(* IEC 61131-3 sources: xPLCCore/codesys_code/Application/COMM_FBs/FB_DataBuffer, 13 files *)

(* ---- FB_DataBuffer.st ---- *)
(*
    FUNCTION_BLOCK FB_DataBuffer

    A re-usable data buffer that operates on an externally provided BYTE array.
    It provides methods for managing a continuous stream of bytes in that external memory.
*)
FUNCTION_BLOCK FB_DataBuffer

VAR
    (* Internal pointers and size information *)
    pBuffer : POINTER TO BYTE; (* Pointer to the start of the external buffer *)
    udiCapacity :DINT;       (* The logical capacity of the external buffer *)
    udiCurrentSize : DINT := 0; (* The current number of valid bytes in the buffer *)
END_VAR
(* =========== IMPLEMENTATION =========== *)

(* ---- get_buffer.st ---- *)
METHOD get_buffer : POINTER TO BYTE
(* =========== IMPLEMENTATION =========== *)
IF pBuffer <> 0 THEN
    get_buffer := pBuffer;
ELSE
    // If the buffer has not been reset, return a NULL pointer.
    get_buffer := 0;
END_IF

(* ---- get_head.st ---- *)
METHOD get_head : POINTER TO BYTE
(* =========== IMPLEMENTATION =========== *)
IF pBuffer <> 0 THEN
    get_head := pBuffer + udiCurrentSize;
ELSE
    // If the buffer has not been reset, return a NULL pointer.
    get_head := 0;
END_IF

(* ---- get_space.st ---- *)
(*
    METHOD get_space : UDINT

    Returns the number of available bytes from the head to the end of the buffer.
*)
METHOD get_space : DINT
(* =========== IMPLEMENTATION =========== *)
IF pBuffer <> 0 THEN
    get_space := udiCapacity - udiCurrentSize;
ELSE
    get_space := 0;
END_IF

(* ---- GetBuffer.st ---- *)
METHOD GetBuffer : POINTER TO BYTE
(* =========== IMPLEMENTATION =========== *)
IF pBuffer <> 0 THEN
    GetBuffer := pBuffer;
ELSE
    // If the buffer has not been reset, return a NULL pointer.
    GetBuffer := 0;
END_IF

(* ---- GetHead.st ---- *)
METHOD GetHead : POINTER TO BYTE
(* =========== IMPLEMENTATION =========== *)
IF pBuffer <> 0 THEN
    GetHead := pBuffer + udiCurrentSize;
ELSE
    // If the buffer has not been reset, return a NULL pointer.
    GetHead := 0;
END_IF

(* ---- GetSpace.st ---- *)
(*
    METHOD GetSpace : UDINT

    Returns the number of available bytes from the head to the end of the buffer.
*)
METHOD GetSpace : DINT
(* =========== IMPLEMENTATION =========== *)
IF pBuffer <> 0 THEN
    GetSpace := udiCapacity - udiCurrentSize;
ELSE
    GetSpace := 0;
END_IF

(* ---- move_left.st ---- *)
METHOD move_left : BOOL
VAR_INPUT
	udiIndex : DINT;
END_VAR
VAR_INST
    udiBytesToMove : DINT;
END_VAR
(* =========== IMPLEMENTATION =========== *)
IF pBuffer <> 0 THEN
    // Check if the consumption index is valid.
    IF udiIndex > 0 AND udiIndex <= udiCurrentSize THEN
        // Calculate the number of bytes remaining after the consumption index.
        udiBytesToMove := udiCurrentSize - udiIndex;

        // Use MEMMOVE to shift the data.
        //MEM.MemMove(pBuffer + udiIndex, pBuffer, UDINT_TO_UINT(udiBytesToMove));//memory overlap is allowed

		MEMUtils.MemCpy(pBuffer, pBuffer + udiIndex, UDINT_TO_UINT(udiBytesToMove));

        // Update the new size of the buffer.
        udiCurrentSize := udiBytesToMove;
    END_IF
END_IF

(* ---- MoveLeft.st ---- *)
METHOD MoveLeft : BOOL
VAR_INPUT
	udiIndex : DINT;
END_VAR
VAR_INST
    udiBytesToMove : DINT;
    diByte         : DINT;
END_VAR
(* =========== IMPLEMENTATION =========== *)
IF pBuffer <> 0 THEN
    // Check if the consumption index is valid.
    IF udiIndex > 0 AND udiIndex <= udiCurrentSize THEN
        // Calculate the number of bytes remaining after the consumption index.
        udiBytesToMove := udiCurrentSize - udiIndex;

        // Shift the rest to the front. Source and destination overlap, and
        // MemCpy does not promise to handle that (review 2026-09-24): copy
        // forward byte by byte, which is correct for a move to the left.
        FOR diByte := 0 TO udiBytesToMove - 1 DO
            pBuffer[diByte] := pBuffer[diByte + udiIndex];
        END_FOR

        // Update the new size of the buffer.
        udiCurrentSize := udiBytesToMove;
    END_IF
END_IF

(* ---- reset_buffer.st ---- *)
METHOD reset_buffer : BOOL
VAR_INPUT
	p_sBuffer : POINTER TO BYTE; (* IN: The address of the external buffer array *)
    udi_Capacity : DINT   ;      (* IN: The total capacity of the external buffer *)
END_VAR
(* =========== IMPLEMENTATION =========== *)
// Store the external buffer's address and capacity internally.
pBuffer := p_sBuffer;
udiCapacity := udi_Capacity;

// Reset the buffer's internal state.
udiCurrentSize := 0;

(* ---- ResetBuffer.st ---- *)
METHOD ResetBuffer : BOOL
VAR_INPUT
	p_sBuffer : POINTER TO BYTE; (* IN: The address of the external buffer array *)
    udi_Capacity : DINT   ;      (* IN: The total capacity of the external buffer *)
END_VAR
(* =========== IMPLEMENTATION =========== *)
// Store the external buffer's address and capacity internally.
pBuffer := p_sBuffer;
udiCapacity := udi_Capacity;

// Reset the buffer's internal state.
udiCurrentSize := 0;

(* ---- write_length.st ---- *)
(*
    METHOD write_length

    Increments the buffer's size by the specified length, effectively "writing" data to it.
    This should be called after an external write operation (e.g., NBS.Read).
*)
METHOD write_length
VAR_INPUT
     udiLength: DINT;
END_VAR
(* =========== IMPLEMENTATION =========== *)
IF pBuffer <> 0 THEN
    // Check for overflow against the logical capacity.
    IF (udiCurrentSize + udiLength) <= udiCapacity THEN
        udiCurrentSize := udiCurrentSize + udiLength;
    ELSE
        // Handle overflow: set size to max capacity.
        udiCurrentSize := udiCapacity;
    END_IF
END_IF

(* ---- WriteLength.st ---- *)
(*
    METHOD WriteLength

    Increments the buffer's size by the specified length, effectively "writing" data to it.
    This should be called after an external write operation (e.g., NBS.Read).
*)
METHOD WriteLength
VAR_INPUT
     udiLength: DINT;
END_VAR
(* =========== IMPLEMENTATION =========== *)
IF pBuffer <> 0 THEN
    // Check for overflow against the logical capacity.
    IF (udiCurrentSize + udiLength) <= udiCapacity THEN
        udiCurrentSize := udiCurrentSize + udiLength;
    ELSE
        // Handle overflow: set size to max capacity.
        udiCurrentSize := udiCapacity;
    END_IF
END_IF
